{attribute 'linkalways'}
{attribute 'qualified_only'}
{attribute 'subsequent'}
{attribute 'pack_mode' := '1'}
VAR_GLOBAL
	Inputs : ST_PLCInputs;
	Outputs : ST_PLCOutputs;
END_VAR

(* stored: Version 1.1.0.1, ProductVersion 3.1.4026.19
   GVL GVL_PLC: Id {6ef7f62b-6fd4-45df-b1d3-ffd68ad3c88b} *)
